// TIA Portal V17 export
// export: Created 2022-07-28T18:02:48.4691933Z, ExportSetting None, DisplayName Totally Integrated Automation Portal, DisplayVersion V17, DisplayName TIA Portal Openness, DisplayVersion V17, DisplayName TIA Portal Teamcenter Gateway, DisplayVersion V17, DisplayName TIA Portal Version Control Interface, DisplayVersion V17, DisplayName TIA Portal Test Suite Advanced, DisplayVersion V17, DisplayName SINAMICS Startdrive Advanced, DisplayVersion V17, DisplayName SINAMICS DCC, DisplayVersion V17, DisplayName SINAMICS Startdrive G130, G150, S120, S150, SINAMICS MV, S210, DisplayVersion V17, DisplayName SINAMICS Startdrive G110M, G120, G120C, G120D, G120P, G115D, DisplayVersion V17, DisplayName STEP 7 Professional, DisplayVersion V17, DisplayName SIMATIC Energy Suite, DisplayVersion V17, DisplayName STEP 7 CFC, DisplayVersion V17, DisplayName STEP 7 Safety, DisplayVersion V17, DisplayName WinCC Advanced / Unified PC, DisplayVersion V17, DisplayName SIMATIC Visualization Architect, DisplayVersion V17
FUNCTION_BLOCK "Lib_FB_AutoMode_CondValves"   // FB5, SCL
{ S7_Optimized_Access := 'TRUE' }
// stored: MemoryReserve 100, SetENOAutomatically false
   VAR_INPUT
      I_Initialization { ExternalAccessible := 'False'; ExternalVisible := 'False'; ExternalWritable := 'False'} : Bool;
   END_VAR
   VAR
      s_EdgeChangePumpVlv1 { ExternalAccessible := 'False'; ExternalVisible := 'False'; ExternalWritable := 'False'} : "Lib_FB_Edge";
      s_EdgeChangePumpVlv2 { ExternalAccessible := 'False'; ExternalVisible := 'False'; ExternalWritable := 'False'} : "Lib_FB_Edge";
      s_EdgeChangePumpVlv3 { ExternalAccessible := 'False'; ExternalVisible := 'False'; ExternalWritable := 'False'} : "Lib_FB_Edge";
      si_PrevPumpVlv1 { S7_SetPoint := 'True'} : Int;
      si_PrevPumpVlv2 { S7_SetPoint := 'True'} : Int := 0;
      si_PrevPumpVlv3 { S7_SetPoint := 'True'} : Int := 0;
   END_VAR
   VAR_TEMP
      ti_ID_Pump1 : Int;
      ti_ID_Pump2 : Int;
      ti_ID_Vlv1 : Int;
      ti_ID_Vlv2 : Int;
      ti_ID_Vlv3 : Int;
      t_DataErr : Bool;   // 1 = Transfer data error occured (ObjDB -> temp, ect)
      tui_NumObjDB : UInt;   // Number of DB for storage object data
      tui_MaxObjects : UInt;   // Max number of objects in plant
      tui_DB_ShiftHMI : UInt;   // Object DB number shift
      tui_DB_ShiftPLC : UInt;   // Object DB number shift
      t_Pump1Any_HMI : DB_ANY;   // Ref to object data
      t_Pump1Var_HMI : Variant;   // Ref to object data
      t_Pump1Any_PLC : DB_ANY;   // Ref to object data
      t_Pump1Var_PLC : Variant;   // Ref to object data
      t_Pump1_HMI : "Lib_UDT_Pump_DS_Base_HMI";   // Object data
      t_Pump1_PLC : "Lib_UDT_Pump_DS_Base_PLC";
      t_Pump1_AutoControl : "Lib_UDT_AutoControl";   // Data for auto control module for current element
      t_Pump2Any_HMI : DB_ANY;   // Ref to object data
      t_Pump2Var_HMI : Variant;   // Ref to object data
      t_Pump2Any_PLC : DB_ANY;   // Ref to object data
      t_Pump2Var_PLC : Variant;   // Ref to object data
      t_Pump2_HMI : "Lib_UDT_Pump_DS_Base_HMI";   // Object data
      t_Pump2_PLC : "Lib_UDT_Pump_DS_Base_PLC";
      t_Pump2_AutoControl : "Lib_UDT_AutoControl";   // Data for auto control module for current element
      t_Vlv1Any_HMI : DB_ANY;   // Ref to object data
      t_Vlv1Var_HMI : Variant;   // Ref to object data
      t_Vlv1Any_PLC : DB_ANY;   // Ref to object data
      t_Vlv1Var_PLC : Variant;   // Ref to object data
      t_Vlv1_HMI : "Lib_UDT_SlideGate_Cond_HMI";   // Object data
      t_Vlv1_PLC : "Lib_UDT_SlideGate_Cond_PLC";
      t_Vlv1_AutoControl : "Lib_UDT_AutoControl";   // Data for auto control module for current element
      t_Vlv2Any_HMI : DB_ANY;   // Ref to object data
      t_Vlv2Var_HMI : Variant;   // Ref to object data
      t_Vlv2Any_PLC : DB_ANY;   // Ref to object data
      t_Vlv2Var_PLC : Variant;   // Ref to object data
      t_Vlv2_HMI : "Lib_UDT_SlideGate_Cond_HMI";   // Object data
      t_Vlv2_PLC : "Lib_UDT_SlideGate_Cond_PLC";
      t_Vlv2_AutoControl : "Lib_UDT_AutoControl";   // Data for auto control module for current element
      t_Vlv3Any_HMI : DB_ANY;   // Ref to object data
      t_Vlv3Var_HMI : Variant;   // Ref to object data
      t_Vlv3Any_PLC : DB_ANY;   // Ref to object data
      t_Vlv3Var_PLC : Variant;   // Ref to object data
      t_Vlv3_HMI : "Lib_UDT_SlideGate_Cond_HMI";   // Object data
      t_Vlv3_PLC : "Lib_UDT_SlideGate_Cond_PLC";
      t_Vlv3_AutoControl : "Lib_UDT_AutoControl";   // Data for auto control module for current element
      t_ReleaseStartPump : Bool;
      t_CmdStartPump : Bool;
      ti_ChoicedPump : Int;
      t_InternalData : "Lib_UDT_Int";   // Internal data
   END_VAR
BEGIN
   REGION Initialization/read data from out DB
       //Set internal data
       "Lib_FC_GenMoto_InitInternal"(#t_InternalData);

       //Set ID for elements in this module
       #ti_ID_Pump1 := 10;
       #ti_ID_Pump2 := 11;
       #ti_ID_Vlv1 := 5;
       #ti_ID_Vlv2 := 6;
       #ti_ID_Vlv3 := 7;

       //Reinit gen data
       #t_DataErr := false;
       #tui_MaxObjects := "D_General_ProgramDATA".ui_MaxObjects;
       #tui_DB_ShiftHMI := "D_General_ProgramDATA".ui_Shift_DB_HMI;
       #tui_DB_ShiftPLC := "D_General_ProgramDATA".ui_Shift_DB_PLC;

       //Read Pump1 data
       //Reinit temp values
       #t_Pump1_HMI := "D_ZeroTypes".Pump_DS_Base_HMI;
       #t_Pump1_PLC := "D_ZeroTypes".Pump_DS_Base_PLC;

       IF #ti_ID_Pump1 >= 0
       THEN
           //Read HMI data
           #tui_NumObjDB := INT_TO_UINT(#ti_ID_Pump1) + #tui_DB_ShiftHMI;
           #t_Pump1Any_HMI := UINT_TO_DB_ANY(#tui_NumObjDB);
           #t_Pump1Var_HMI := DB_ANY_TO_VARIANT(in := #t_Pump1Any_HMI, err => #t_InternalData.i_Tmp);

           //If DB exist and convertion without error
           IF #t_InternalData.i_Tmp = 0
           THEN
               VariantGet(SRC := #t_Pump1Var_HMI,
                          DST => #t_Pump1_HMI);
           ELSE
               #t_DataErr := true;
           END_IF;

           //Read PLC data
           #tui_NumObjDB := INT_TO_UINT(#ti_ID_Pump1) + #tui_DB_ShiftPLC;
           #t_Pump1Any_PLC := UINT_TO_DB_ANY(#tui_NumObjDB);
           #t_Pump1Var_PLC := DB_ANY_TO_VARIANT(in := #t_Pump1Any_PLC, err => #t_InternalData.i_Tmp);

           //If DB exist and convertion without error
           IF #t_InternalData.i_Tmp = 0
           THEN
               VariantGet(SRC := #t_Pump1Var_PLC,
                          DST => #t_Pump1_PLC);
           ELSE
               #t_DataErr := true;
           END_IF;
       ELSE
           #t_DataErr := true;
       END_IF;

       //Read general info data
       #t_Pump1_AutoControl := "DB_AutoControl_arr".AutoControl_arr[#tui_MaxObjects];
       CASE #ti_ID_Pump1 OF
           0..999:  // ID of element in range
               #t_Pump1_AutoControl := "DB_AutoControl_arr".AutoControl_arr[#ti_ID_Pump1];
           ELSE
               ;
       END_CASE;

       //Read Pump2 data
       //Reinit temp values
       #t_Pump2_HMI := "D_ZeroTypes".Pump_DS_Base_HMI;
       #t_Pump2_PLC := "D_ZeroTypes".Pump_DS_Base_PLC;

       IF #ti_ID_Pump2 >= 0
       THEN
           //Read HMI data
           #tui_NumObjDB := INT_TO_UINT(#ti_ID_Pump2) + #tui_DB_ShiftHMI;
           #t_Pump2Any_HMI := UINT_TO_DB_ANY(#tui_NumObjDB);
           #t_Pump2Var_HMI := DB_ANY_TO_VARIANT(in := #t_Pump2Any_HMI, err => #t_InternalData.i_Tmp);

           //If DB exist and convertion without error
           IF #t_InternalData.i_Tmp = 0
           THEN
               VariantGet(SRC := #t_Pump2Var_HMI,
                          DST => #t_Pump2_HMI);
           ELSE
               #t_DataErr := true;
           END_IF;

           //Read PLC data
           #tui_NumObjDB := INT_TO_UINT(#ti_ID_Pump2) + #tui_DB_ShiftPLC;
           #t_Pump2Any_PLC := UINT_TO_DB_ANY(#tui_NumObjDB);
           #t_Pump2Var_PLC := DB_ANY_TO_VARIANT(in := #t_Pump2Any_PLC, err => #t_InternalData.i_Tmp);

           //If DB exist and convertion without error
           IF #t_InternalData.i_Tmp = 0
           THEN
               VariantGet(SRC := #t_Pump2Var_PLC,
                          DST => #t_Pump2_PLC);
           ELSE
               #t_DataErr := true;
           END_IF;
       ELSE
           #t_DataErr := true;
       END_IF;

       //Read general info data
       #t_Pump2_AutoControl := "DB_AutoControl_arr".AutoControl_arr[#tui_MaxObjects];
       CASE #ti_ID_Pump2 OF
           0..999:  // ID of element in range
               #t_Pump2_AutoControl := "DB_AutoControl_arr".AutoControl_arr[#ti_ID_Pump2];
           ELSE
               ;
       END_CASE;

       //Read Valve1 data
       //Reinit temp values
       #t_Vlv1_HMI := "D_ZeroTypes".SlideGate_Cond_HMI;
       #t_Vlv1_PLC := "D_ZeroTypes".SlideGate_Cond_PLC;

       IF #ti_ID_Vlv1 >= 0
       THEN
           //Read HMI data
           #tui_NumObjDB := INT_TO_UINT(#ti_ID_Vlv1) + #tui_DB_ShiftHMI;
           #t_Vlv1Any_HMI := UINT_TO_DB_ANY(#tui_NumObjDB);
           #t_Vlv1Var_HMI := DB_ANY_TO_VARIANT(in := #t_Vlv1Any_HMI, err => #t_InternalData.i_Tmp);

           //If DB exist and convertion without error
           IF #t_InternalData.i_Tmp = 0
           THEN
               VariantGet(SRC := #t_Vlv1Var_HMI,
                          DST => #t_Vlv1_HMI);
           ELSE
               #t_DataErr := true;
           END_IF;

           //Read PLC data
           #tui_NumObjDB := INT_TO_UINT(#ti_ID_Vlv1) + #tui_DB_ShiftPLC;
           #t_Vlv1Any_PLC := UINT_TO_DB_ANY(#tui_NumObjDB);
           #t_Vlv1Var_PLC := DB_ANY_TO_VARIANT(in := #t_Vlv1Any_PLC, err => #t_InternalData.i_Tmp);

           //If DB exist and convertion without error
           IF #t_InternalData.i_Tmp = 0
           THEN
               VariantGet(SRC := #t_Vlv1Var_PLC,
                          DST => #t_Vlv1_PLC);
           ELSE
               #t_DataErr := true;
           END_IF;
       ELSE
           #t_DataErr := true;
       END_IF;

       //Read general info data
       #t_Vlv1_AutoControl := "DB_AutoControl_arr".AutoControl_arr[#tui_MaxObjects];
       CASE #ti_ID_Vlv1 OF
           0..999:  // ID of element in range
               #t_Vlv1_AutoControl := "DB_AutoControl_arr".AutoControl_arr[#ti_ID_Vlv1];
           ELSE
               ;
       END_CASE;

       //Read Valve2 data
       //Reinit temp values
       #t_Vlv2_HMI := "D_ZeroTypes".SlideGate_Cond_HMI;
       #t_Vlv2_PLC := "D_ZeroTypes".SlideGate_Cond_PLC;

       IF #ti_ID_Vlv2 >= 0
       THEN
           //Read HMI data
           #tui_NumObjDB := INT_TO_UINT(#ti_ID_Vlv2) + #tui_DB_ShiftHMI;
           #t_Vlv2Any_HMI := UINT_TO_DB_ANY(#tui_NumObjDB);
           #t_Vlv2Var_HMI := DB_ANY_TO_VARIANT(in := #t_Vlv2Any_HMI, err => #t_InternalData.i_Tmp);

           //If DB exist and convertion without error
           IF #t_InternalData.i_Tmp = 0
           THEN
               VariantGet(SRC := #t_Vlv2Var_HMI,
                          DST => #t_Vlv2_HMI);
           ELSE
               #t_DataErr := true;
           END_IF;

           //Read PLC data
           #tui_NumObjDB := INT_TO_UINT(#ti_ID_Vlv2) + #tui_DB_ShiftPLC;
           #t_Vlv2Any_PLC := UINT_TO_DB_ANY(#tui_NumObjDB);
           #t_Vlv2Var_PLC := DB_ANY_TO_VARIANT(in := #t_Vlv2Any_PLC, err => #t_InternalData.i_Tmp);

           //If DB exist and convertion without error
           IF #t_InternalData.i_Tmp = 0
           THEN
               VariantGet(SRC := #t_Vlv2Var_PLC,
                          DST => #t_Vlv2_PLC);
           ELSE
               #t_DataErr := true;
           END_IF;
       ELSE
           #t_DataErr := true;
       END_IF;

       //Read general info data
       #t_Vlv2_AutoControl := "DB_AutoControl_arr".AutoControl_arr[#tui_MaxObjects];
       CASE #ti_ID_Vlv2 OF
           0..999:  // ID of element in range
               #t_Vlv2_AutoControl := "DB_AutoControl_arr".AutoControl_arr[#ti_ID_Vlv2];
           ELSE
               ;
       END_CASE;

       //Read Valve3 data
       //Reinit temp values
       #t_Vlv3_HMI := "D_ZeroTypes".SlideGate_Cond_HMI;
       #t_Vlv3_PLC := "D_ZeroTypes".SlideGate_Cond_PLC;

       IF #ti_ID_Vlv3 >= 0
       THEN
           //Read HMI data
           #tui_NumObjDB := INT_TO_UINT(#ti_ID_Vlv3) + #tui_DB_ShiftHMI;
           #t_Vlv3Any_HMI := UINT_TO_DB_ANY(#tui_NumObjDB);
           #t_Vlv3Var_HMI := DB_ANY_TO_VARIANT(in := #t_Vlv3Any_HMI, err => #t_InternalData.i_Tmp);

           //If DB exist and convertion without error
           IF #t_InternalData.i_Tmp = 0
           THEN
               VariantGet(SRC := #t_Vlv3Var_HMI,
                          DST => #t_Vlv3_HMI);
           ELSE
               #t_DataErr := true;
           END_IF;

           //Read PLC data
           #tui_NumObjDB := INT_TO_UINT(#ti_ID_Vlv3) + #tui_DB_ShiftPLC;
           #t_Vlv3Any_PLC := UINT_TO_DB_ANY(#tui_NumObjDB);
           #t_Vlv3Var_PLC := DB_ANY_TO_VARIANT(in := #t_Vlv3Any_PLC, err => #t_InternalData.i_Tmp);

           //If DB exist and convertion without error
           IF #t_InternalData.i_Tmp = 0
           THEN
               VariantGet(SRC := #t_Vlv3Var_PLC,
                          DST => #t_Vlv3_PLC);
           ELSE
               #t_DataErr := true;
           END_IF;
       ELSE
           #t_DataErr := true;
       END_IF;

       //Read general info data
       #t_Vlv3_AutoControl := "DB_AutoControl_arr".AutoControl_arr[#tui_MaxObjects];
       CASE #ti_ID_Vlv3 OF
           0..999:  // ID of element in range
               #t_Vlv3_AutoControl := "DB_AutoControl_arr".AutoControl_arr[#ti_ID_Vlv3];
           ELSE
               ;
       END_CASE;

   END_REGION
   //---------------------------------------------------------------
   //---------------------------------------------------------------
   REGION Catch if choiced pump was changed
       //Set previous pump durring initialization
       IF #I_Initialization
       THEN
           #t_Vlv1_HMI.Config.i_ChoicedPump := 1;
           #t_Vlv2_HMI.Config.i_ChoicedPump := 1;
           #t_Vlv3_HMI.Config.i_ChoicedPump := 1;

           #si_PrevPumpVlv1 := #t_Vlv1_HMI.Config.i_ChoicedPump;
           #si_PrevPumpVlv2 := #t_Vlv2_HMI.Config.i_ChoicedPump;
           #si_PrevPumpVlv3 := #t_Vlv3_HMI.Config.i_ChoicedPump;
       END_IF;

       //Catch change of choiced pump
       #s_EdgeChangePumpVlv1(IB_Initialisation:=#I_Initialization,
                             IB_Input:=#si_PrevPumpVlv1 <> #t_Vlv1_HMI.Config.i_ChoicedPump,
                             QB_EdgePos=> #s_EdgeChangePumpVlv1.QB_EdgePos);

       #s_EdgeChangePumpVlv2(IB_Initialisation := #I_Initialization,
                             IB_Input := #si_PrevPumpVlv2 <> #t_Vlv2_HMI.Config.i_ChoicedPump,
                             QB_EdgePos => #s_EdgeChangePumpVlv2.QB_EdgePos);

       #s_EdgeChangePumpVlv3(IB_Initialisation := #I_Initialization,
                             IB_Input := #si_PrevPumpVlv3 <> #t_Vlv3_HMI.Config.i_ChoicedPump,
                             QB_EdgePos => #s_EdgeChangePumpVlv3.QB_EdgePos);

       //Rewrite others if in some one change occured
       IF #s_EdgeChangePumpVlv1.QB_EdgePos
       THEN
           #t_Vlv2_HMI.Config.i_ChoicedPump := #t_Vlv1_HMI.Config.i_ChoicedPump;
           #t_Vlv3_HMI.Config.i_ChoicedPump := #t_Vlv1_HMI.Config.i_ChoicedPump;
       END_IF;
       IF #s_EdgeChangePumpVlv2.QB_EdgePos
       THEN
           #t_Vlv1_HMI.Config.i_ChoicedPump := #t_Vlv2_HMI.Config.i_ChoicedPump;
           #t_Vlv3_HMI.Config.i_ChoicedPump := #t_Vlv2_HMI.Config.i_ChoicedPump;
       END_IF;
       IF #s_EdgeChangePumpVlv3.QB_EdgePos
       THEN
           #t_Vlv2_HMI.Config.i_ChoicedPump := #t_Vlv3_HMI.Config.i_ChoicedPump;
           #t_Vlv1_HMI.Config.i_ChoicedPump := #t_Vlv3_HMI.Config.i_ChoicedPump;
       END_IF;

       #si_PrevPumpVlv1 := #t_Vlv1_HMI.Config.i_ChoicedPump;
       #si_PrevPumpVlv2 := #t_Vlv2_HMI.Config.i_ChoicedPump;
       #si_PrevPumpVlv3 := #t_Vlv3_HMI.Config.i_ChoicedPump;

       //Set choiced pump
       #ti_ChoicedPump := #t_Vlv1_HMI.Config.i_ChoicedPump;
   END_REGION
   //---------------------------------------------------------------
   //---------------------------------------------------------------
   REGION Conditions for run pump in auto mode and start them in auto
       #t_ReleaseStartPump := false;

       CASE #ti_ChoicedPump OF
           1:  // Choiced pump PR46.1
               #t_ReleaseStartPump := #t_Pump1_PLC.Mode.Auto
               AND #t_Pump1_PLC.State.Ready;
           2:  // Choiced pump PR46.2
               #t_ReleaseStartPump := #t_Pump2_PLC.Mode.Auto
               AND #t_Pump2_PLC.State.Ready;
           ELSE
               #t_ReleaseStartPump := false;
       END_CASE;

       #t_CmdStartPump := ((#t_Vlv1_PLC.State.Opened
       AND #t_Vlv1_AutoControl.Mode.Auto)
       OR (#t_Vlv2_PLC.State.Opened
       AND #t_Vlv2_AutoControl.Mode.Auto)
       OR (#t_Vlv3_PLC.State.Opened
       AND #t_Vlv3_AutoControl.Mode.Auto))
       AND #t_ReleaseStartPump;

       CASE #ti_ChoicedPump OF
           1:  // Choiced pump PR46.1
               #t_Pump1_AutoControl.CTW := dw#16#0;
               #t_Pump2_AutoControl.CTW := dw#16#0;

               #t_Pump1_AutoControl.CTW.%X0 := #t_CmdStartPump;
               #t_Pump1_AutoControl.StatusGen.Release := #t_ReleaseStartPump;

               #t_Vlv1_PLC.State.PumpIsAuto := #t_Pump1_PLC.Mode.Auto;
               #t_Vlv1_PLC.State.PumpIsReady := #t_Pump1_PLC.State.Ready;
               #t_Vlv1_PLC.State.PumpIsRunning := #t_Pump1_PLC.State.Run;

               #t_Vlv2_PLC.State.PumpIsAuto := #t_Pump1_PLC.Mode.Auto;
               #t_Vlv2_PLC.State.PumpIsReady := #t_Pump1_PLC.State.Ready;
               #t_Vlv2_PLC.State.PumpIsRunning := #t_Pump1_PLC.State.Run;

               #t_Vlv3_PLC.State.PumpIsAuto := #t_Pump1_PLC.Mode.Auto;
               #t_Vlv3_PLC.State.PumpIsReady := #t_Pump1_PLC.State.Ready;
               #t_Vlv3_PLC.State.PumpIsRunning := #t_Pump1_PLC.State.Run;

           2:  // Choiced pump PR46.2
               #t_Pump1_AutoControl.CTW := dw#16#0;
               #t_Pump2_AutoControl.CTW := dw#16#0;

               #t_Pump2_AutoControl.CTW.%X0 := #t_CmdStartPump;
               #t_Pump2_AutoControl.StatusGen.Release := #t_ReleaseStartPump;

               #t_Vlv1_PLC.State.PumpIsAuto := #t_Pump2_PLC.Mode.Auto;
               #t_Vlv1_PLC.State.PumpIsReady := #t_Pump2_PLC.State.Ready;
               #t_Vlv1_PLC.State.PumpIsRunning := #t_Pump2_PLC.State.Run;

               #t_Vlv2_PLC.State.PumpIsAuto := #t_Pump2_PLC.Mode.Auto;
               #t_Vlv2_PLC.State.PumpIsReady := #t_Pump2_PLC.State.Ready;
               #t_Vlv2_PLC.State.PumpIsRunning := #t_Pump2_PLC.State.Run;

               #t_Vlv3_PLC.State.PumpIsAuto := #t_Pump2_PLC.Mode.Auto;
               #t_Vlv3_PLC.State.PumpIsReady := #t_Pump2_PLC.State.Ready;
               #t_Vlv3_PLC.State.PumpIsRunning := #t_Pump2_PLC.State.Run;
           ELSE
               #t_Vlv1_PLC.State.PumpIsAuto := false;
               #t_Vlv1_PLC.State.PumpIsReady := false;
               #t_Vlv1_PLC.State.PumpIsRunning := false;

               #t_Vlv2_PLC.State.PumpIsAuto := false;
               #t_Vlv2_PLC.State.PumpIsReady := false;
               #t_Vlv2_PLC.State.PumpIsRunning := false;

               #t_Vlv3_PLC.State.PumpIsAuto := false;
               #t_Vlv3_PLC.State.PumpIsReady := false;
               #t_Vlv3_PLC.State.PumpIsRunning := false;
       END_CASE;
   END_REGION
   //---------------------------------------------------------------
   //---------------------------------------------------------------
   REGION Write data to modules

       //Write Pump1 data
       //DB num 
       IF #ti_ID_Pump1 >= 0
           AND NOT #t_DataErr
       THEN
           //Write HMI data
           VariantPut(SRC := #t_Pump1_HMI,
                      DST := #t_Pump1Var_HMI);

           //Write PLC data
           VariantPut(SRC := #t_Pump1_PLC,
                      DST := #t_Pump1Var_PLC);
       ELSE
           #t_DataErr := true;
       END_IF;

       //Write general info data
       CASE #ti_ID_Pump1 OF
           0..999:  // ID of element in range
               "DB_AutoControl_arr".AutoControl_arr[#ti_ID_Pump1] := #t_Pump1_AutoControl;
           ELSE
               ;
       END_CASE;

       //Write Pump2 data
       //DB num 
       IF #ti_ID_Pump2 >= 0
           AND NOT #t_DataErr
       THEN
           //Write HMI data
           VariantPut(SRC := #t_Pump2_HMI,
                      DST := #t_Pump2Var_HMI);

           //Write PLC data
           VariantPut(SRC := #t_Pump2_PLC,
                      DST := #t_Pump2Var_PLC);
       ELSE
           #t_DataErr := true;
       END_IF;

       //Write general info data
       CASE #ti_ID_Pump2 OF
           0..999:  // ID of element in range
               "DB_AutoControl_arr".AutoControl_arr[#ti_ID_Pump2] := #t_Pump2_AutoControl;
           ELSE
               ;
       END_CASE;

       //Write Vlv1 data
       //DB num 
       IF #ti_ID_Vlv1 >= 0
           AND NOT #t_DataErr
       THEN
           //Write HMI data
           VariantPut(SRC := #t_Vlv1_HMI,
                      DST := #t_Vlv1Var_HMI);

           //Write PLC data
           VariantPut(SRC := #t_Vlv1_PLC,
                      DST := #t_Vlv1Var_PLC);
       ELSE
           #t_DataErr := true;
       END_IF;

       //Write general info data
       CASE #ti_ID_Vlv1 OF
           0..999:  // ID of element in range
               "DB_AutoControl_arr".AutoControl_arr[#ti_ID_Vlv1] := #t_Vlv1_AutoControl;
           ELSE
               ;
       END_CASE;

       //Write Vlv2 data
       //DB num 
       IF #ti_ID_Vlv2 >= 0
           AND NOT #t_DataErr
       THEN
           //Write HMI data
           VariantPut(SRC := #t_Vlv2_HMI,
                      DST := #t_Vlv2Var_HMI);

           //Write PLC data
           VariantPut(SRC := #t_Vlv2_PLC,
                      DST := #t_Vlv2Var_PLC);
       ELSE
           #t_DataErr := true;
       END_IF;

       //Write general info data
       CASE #ti_ID_Vlv2 OF
           0..999:  // ID of element in range
               "DB_AutoControl_arr".AutoControl_arr[#ti_ID_Vlv2] := #t_Vlv2_AutoControl;
           ELSE
               ;
       END_CASE;

       //Write Vlv3 data
       //DB num 
       IF #ti_ID_Vlv3 >= 0
           AND NOT #t_DataErr
       THEN
           //Write HMI data
           VariantPut(SRC := #t_Vlv3_HMI,
                      DST := #t_Vlv3Var_HMI);

           //Write PLC data
           VariantPut(SRC := #t_Vlv3_PLC,
                      DST := #t_Vlv3Var_PLC);
       ELSE
           #t_DataErr := true;
       END_IF;

       //Write general info data
       CASE #ti_ID_Vlv3 OF
           0..999:  // ID of element in range
               "DB_AutoControl_arr".AutoControl_arr[#ti_ID_Vlv3] := #t_Vlv3_AutoControl;
           ELSE
               ;
       END_CASE;

   END_REGION
   //---------------------------------------------------------------
   //---------------------------------------------------------------
END_FUNCTION_BLOCK
